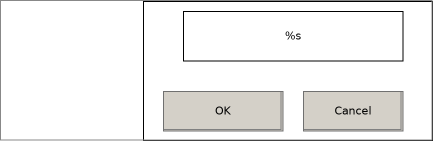
VISUALIZATION DialogTest  // 433x141
VAR_INPUT
	sText: string;
END_VAR
    Rectangle (143,1 290x140)
    Rectangle (183,11 220x50), "%s", text variable: sText
    Button (163,91 120x40), "OK"
        OnDialogClosed: execute { P_Dialog.bVisible:=TRUE; P_Dialog.bClose:=TRUE; }
        OnMouseClick: CloseDialog Dialog=DialogTest, Result=OK, NumpadKeypadSet=True
    Button (303,91 100x40), "Cancel"
        OnDialogClosed: execute { P_Dialog.bVisible:=TRUE; P_Dialog.bClose:=TRUE; }
        OnMouseClick: CloseDialog Dialog=DialogTest, Result=Cancel, NumpadKeypadSet=True
END_VISUALIZATION

(* stored: Version 1.1.0.1, ProductVersion 3.1.4024.12
   Visu DialogTest: Id {0500f354-c7ac-4b40-aef5-420d696610dc} *)
